(* CODESYS project plc_chalet_base.library
   Title: CHALET_BaseComponents
   Version: 3.6.9
   Placeholder: CHALET_BaseComponents
   Company: Beckhoff CH

Project tree, tasks and I/O mapping:
  libraries: Tc2_EtherCAT, * (Beckhoff Automation GmbH); Tc2_Standard, * (Beckhoff Automation GmbH); Tc2_System, * (Beckhoff Automation GmbH); Tc2_Utilities, * (Beckhoff Automation GmbH); Tc3_EventLogger, * (Beckhoff Automation GmbH); Tc3_Module, * (Beckhoff Automation GmbH)
  COMPONENTs/
    CoE-Access/
      internal/
        function block FB_CoE_Base [ST]: cbBufLen, Index, pSrcBuf, SubIndex, Error, FB_init, ReadDone, Update, WriteDone
        interface I_AdsAddr: NetId, Port
      function block FB_CoE_BOOL [ST]: cbBufLen, pSrcBuf, Value
      function block FB_CoE_BYTE [ST]: cbBufLen, pSrcBuf, Value
      function block FB_CoE_Connection [ST]: Mapped, NetId, Port
      function block FB_CoE_UDINT [ST]: cbBufLen, pSrcBuf, Value
      function block FB_CoE_UINT [ST]: cbBufLen, pSrcBuf, Value
    EtherCatDiag/
      Subobject/
        data type E_EtherCatState
        function block FB_EtherCatSlaveDiag [ST]: AlarmHandling, DeviceAmsAddr, DeviceType, Name, SetConfig, State, StateBits, Update
        interface I_EtherCatSlaveDiag: DeviceAmsAddr, DeviceType, Name, State, StateBits
      function block FB_EtherCatMasterDiag [ST]: Initialize, Initialized, ListOfDevices, Mapped, NumerOfDevice, Update
      data type ST_XtsMotorEtherCatDiag
    Feedback/
      function block FB_CH_Feedback [ST]: ActiveCommand, Busy, Done, Error, ErrorId, FB_init, HR, LastCommandAccepted, UpdateEventlogger
      interface I_CH_Feedback: ActiveCommand, Busy, Done, Error, ErrorId, HR, LastCommandAccepted
    HR/
      function CheckNotOk [ST]
      function CheckOk [ST]
      function GetMostSignificant [ST]
    List/
      CD_CH_List
      function block FB_CH_List [ST]: Content, FindLUID, FindOID, FindOIDString, LUIDInList, OIDInList, ResetIterator, RestoreIterator, AddList, Clear, Duplicate, Initialize, IsEmpty, IsFull, Size, Update, AddObject, GetNextObject, GetRandomObject, HasNextObject, ObjectInList, RemoveAllDuplicateObjects, RemoveObject, GetObjectWithHighestNumber, GetObjectWithLowestNumber, Sort
      interface I_CH_List: Content, FindLUID, FindOID, FindOIDString, LUIDInList, OIDInList, ResetIterator, RestoreIterator, IsEmpty, IsFull, Size, GetNextObject, GetRandomObject, HasNextObject, ObjectInList, RemoveAllDuplicateObjects, GetObjectWithHighestNumber, GetObjectWithLowestNumber
      interface I_CH_List_Dublicate: Content
    Object/
      CD_CH_Object
      function block FB_CH_Object [ST]: FB_init, Initialize, LUID, OID, SortOrderInList, TaskIndex, Update
      interface I_CH_Object: Initialize, LUID, OID, SortOrderInList, Update
    function F_Convert32InPastTo64Bit [ST]
  CONSTANTs/
    data type E_Colors_ARGB
    global variables GVL_Datatypes
  global variables BaseParameterlist
  00000000-0000-0000-0000-000000000000|LICENSE.md
  LICENSE.md
*)

// COMPONENTs/EtherCatDiag/Subobject/E_EtherCatState
{attribute 'qualified_only'}
{attribute 'strict'}
{attribute 'to_string'}
TYPE E_EtherCatState :
(
	Unknown,
	Init,
	PreOp,
	BootStrap,
	SafeOp,
	Op,
	Disabled,
	Error
) := Unknown ;
END_TYPE

// COMPONENTs/EtherCatDiag/ST_XtsMotorEtherCatDiag
TYPE ST_XtsMotorEtherCatDiag :
STRUCT
	fbSource : FB_TcSourceInfo;
	fbAlarmNotInOpMode : FB_TcAlarm;
	fbAlarmNoCommunication : FB_TcAlarm;
	
	fbGetSlaveState : FB_EcGetSlaveState;
	nLastState : BYTE;
END_STRUCT
END_TYPE

// CONSTANTs/E_Colors_ARGB
{attribute 'qualified_only'}
{attribute 'strict'}
{attribute 'to_string'}
TYPE E_Colors_ARGB : (
        Darkred              := 16#FF8B0000, // rgb(139,0,0)
        Brown                := 16#FFA52A2A, // rgb(165,42,42)
        Firebrick            := 16#FFB22222, // rgb(178,34,34)
        Crimson              := 16#FFDC143C, // rgb(220,20,60)
        Red                  := 16#FFFF0000, // rgb(255,0,0)
        Tomato               := 16#FFFF6347, // rgb(255,99,71)
        Coral                := 16#FFFF7F50, // rgb(255,127,80)
        Indianred            := 16#FFCD5C5C, // rgb(205,92,92)
        Lightcoral           := 16#FFF08080, // rgb(240,128,128)
        Darksalmon           := 16#FFE9967A, // rgb(233,150,122)
        Salmon               := 16#FFFA8072, // rgb(250,128,114)
        Lightsalmon          := 16#FFFFA07A, // rgb(255,160,122)
        Orangered            := 16#FFFF4500, // rgb(255,69,0)
        Darkorange           := 16#FFFF8C00, // rgb(255,140,0)
        Orange               := 16#FFFFA500, // rgb(255,165,0)
        Gold                 := 16#FFFFD700, // rgb(255,215,0)
        Darkgoldenrod        := 16#FFB8860B, // rgb(184,134,11)
        Goldenrod            := 16#FFDAA520, // rgb(218,165,32)
        Palegoldenrod        := 16#FFEEE8AA, // rgb(238,232,170)
        Darkkhaki            := 16#FFBDB76B, // rgb(189,183,107)
        Khaki                := 16#FFF0E68C, // rgb(240,230,140)
        Olive                := 16#FF808000, // rgb(128,128,0)
        Yellow               := 16#FFFFFF00, // rgb(255,255,0)
        Yellowgreen          := 16#FF9ACD32, // rgb(154,205,50)
        Darkolivegreen       := 16#FF556B2F, // rgb(85,107,47)
        Olivedrab            := 16#FF6B8E23, // rgb(107,142,35)
        Lawngreen            := 16#FF7CFC00, // rgb(124,252,0)
        Chartreuse           := 16#FF7FFF00, // rgb(127,255,0)
        Greenyellow          := 16#FFADFF2F, // rgb(173,255,47)
        Darkgreen            := 16#FF006400, // rgb(0,100,0)
        Green                := 16#FF008000, // rgb(0,128,0)
        Forestgreen          := 16#FF228B22, // rgb(34,139,34)
        Lime                 := 16#FF00FF00, // rgb(0,255,0)
        Limegreen            := 16#FF32CD32, // rgb(50,205,50)
        Lightgreen           := 16#FF90EE90, // rgb(144,238,144)
        Palegreen            := 16#FF98FB98, // rgb(152,251,152)
        Darkseagreen         := 16#FF8FBC8F, // rgb(143,188,143)
        Mediumspringgreen    := 16#FF00FA9A, // rgb(0,250,154)
        Springgreen          := 16#FF00FF7F, // rgb(0,255,127)
        Seagreen             := 16#FF2E8B57, // rgb(46,139,87)
        Mediumaquamarine     := 16#FF66CDAA, // rgb(102,205,170)
        Mediumseagreen       := 16#FF3CB371, // rgb(60,179,113)
        Lightseagreen        := 16#FF20B2AA, // rgb(32,178,170)
        Darkslategray        := 16#FF2F4F4F, // rgb(47,79,79)
        Teal                 := 16#FF008080, // rgb(0,128,128)
        Darkcyan             := 16#FF008B8B, // rgb(0,139,139)
        Aqua                 := 16#FF00FFFF, // rgb(0,255,255)
        Lightcyan            := 16#FFE0FFFF, // rgb(224,255,255)
        Darkturquoise        := 16#FF00CED1, // rgb(0,206,209)
        Turquoise            := 16#FF40E0D0, // rgb(64,224,208)
        Mediumturquoise      := 16#FF48D1CC, // rgb(72,209,204)
        Paleturquoise        := 16#FFAFEEEE, // rgb(175,238,238)
        Aquamarine           := 16#FF7FFFD4, // rgb(127,255,212)
        Powderblue           := 16#FFB0E0E6, // rgb(176,224,230)
        Cadetblue            := 16#FF5F9EA0, // rgb(95,158,160)
        Steelblue            := 16#FF4682B4, // rgb(70,130,180)
        Cornflowerblue       := 16#FF6495ED, // rgb(100,149,237)
        Deepskyblue          := 16#FF00BFFF, // rgb(0,191,255)
        Dodgerblue           := 16#FF1E90FF, // rgb(30,144,255)
        Lightblue            := 16#FFADD8E6, // rgb(173,216,230)
        Skyblue              := 16#FF87CEEB, // rgb(135,206,235)
        Lightskyblue         := 16#FF87CEFA, // rgb(135,206,250)
        Midnightblue         := 16#FF191970, // rgb(25,25,112)
        Navy                 := 16#FF000080, // rgb(0,0,128)
        Darkblue             := 16#FF00008B, // rgb(0,0,139)
        Mediumblue           := 16#FF0000CD, // rgb(0,0,205)
        Blue                 := 16#FF0000FF, // rgb(0,0,255)
        Royalblue            := 16#FF4169E1, // rgb(65,105,225)
        Blueviolet           := 16#FF8A2BE2, // rgb(138,43,226)
        Indigo               := 16#FF4B0082, // rgb(75,0,130)
        Darkslateblue        := 16#FF483D8B, // rgb(72,61,139)
        Slateblue            := 16#FF6A5ACD, // rgb(106,90,205)
        Mediumslateblue      := 16#FF7B68EE, // rgb(123,104,238)
        Mediumpurple         := 16#FF9370DB, // rgb(147,112,219)
        Darkmagenta          := 16#FF8B008B, // rgb(139,0,139)
        Darkviolet           := 16#FF9400D3, // rgb(148,0,211)
        Darkorchid           := 16#FF9932CC, // rgb(153,50,204)
        Mediumorchid         := 16#FFBA55D3, // rgb(186,85,211)
        Purple               := 16#FF800080, // rgb(128,0,128)
        Thistle              := 16#FFD8BFD8, // rgb(216,191,216)
        Plum                 := 16#FFDDA0DD, // rgb(221,160,221)
        Violet               := 16#FFEE82EE, // rgb(238,130,238)
        Magenta              := 16#FFFF00FF, // rgb(255,0,255)
        Orchid               := 16#FFDA70D6, // rgb(218,112,214)
        Mediumvioletred      := 16#FFC71585, // rgb(199,21,133)
        Palevioletred        := 16#FFDB7093, // rgb(219,112,147)
        Deeppink             := 16#FFFF1493, // rgb(255,20,147)
        Hotpink              := 16#FFFF69B4, // rgb(255,105,180)
        Lightpink            := 16#FFFFB6C1, // rgb(255,182,193)
        Pink                 := 16#FFFFC0CB, // rgb(255,192,203)
        Antiquewhite         := 16#FFFAEBD7, // rgb(250,235,215)
        Beige                := 16#FFF5F5DC, // rgb(245,245,220)
        Bisque               := 16#FFFFE4C4, // rgb(255,228,196)
        Blanchedalmond       := 16#FFFFEBCD, // rgb(255,235,205)
        Wheat                := 16#FFF5DEB3, // rgb(245,222,179)
        Cornsilk             := 16#FFFFF8DC, // rgb(255,248,220)
        Lemonchiffon         := 16#FFFFFACD, // rgb(255,250,205)
        LightGoldenRodYellow := 16#FFFAFAD2, // rgb(250,250,210)
        LightYellow          := 16#FFFFFFE0, // rgb(255,255,224)
        SaddleBrown          := 16#FF8B4513, // rgb(139,69,19)
        Sienna               := 16#FFA0522D, // rgb(160,82,45)
        Chocolate            := 16#FFD2691E, // rgb(210,105,30)
        Peru                 := 16#FFCD853F, // rgb(205,133,63)
        SandyBrown           := 16#FFF4A460, // rgb(244,164,96)
        BurlyWood            := 16#FFDEB887, // rgb(222,184,135)
        RosyBrown            := 16#FFBC8F8F, // rgb(188,143,143)
        Moccasin             := 16#FFFFE4B5, // rgb(255,228,181)
        NavajoWhite          := 16#FFFFDEAD, // rgb(255,222,173)
        PeachPuff            := 16#FFFFDAB9, // rgb(255,218,185)
        MistyRose            := 16#FFFFE4E1, // rgb(255,228,225)
        LavenderBlush        := 16#FFFFF0F5, // rgb(255,240,245)
        Linen                := 16#FFFAF0E6, // rgb(250,240,230)
        OldLace              := 16#FFFDF5E6, // rgb(253,245,230)
        PapayaWhip           := 16#FFFFEFD5, // rgb(255,239,213)
        Seashell             := 16#FFFFF5EE, // rgb(255,245,238)
        MintCream            := 16#FFF5FFFA, // rgb(245,255,250)
        SlateGray            := 16#FF708090, // rgb(112,128,144)
        LightSlateGray       := 16#FF778899, // rgb(119,136,153)
        LightSteelBlue       := 16#FFB0C4DE, // rgb(176,196,222)
        Lavender             := 16#FFE6E6FA, // rgb(230,230,250)
        FloralWhite          := 16#FFFFFAF0, // rgb(255,250,240)
        AliceBlue            := 16#FFF0F8FF, // rgb(240,248,255)
        GhostWhite           := 16#FFF8F8FF, // rgb(248,248,255)
        HoneyDew             := 16#FFF0FFF0, // rgb(240,255,240)
        Ivory                := 16#FFFFFFF0, // rgb(255,255,240)
        Azure                := 16#FFF0FFFF, // rgb(240,255,255)
        Snow                 := 16#FFFFFAFA, // rgb(255,250,250)
        Black                := 16#FF000000, // rgb(0,0,0)
        DimGray              := 16#FF696969, // rgb(105,105,105)
        Gray                 := 16#FF808080, // rgb(128,128,128)
        DarkGray             := 16#FFA9A9A9, // rgb(169,169,169)
        Silver               := 16#FFC0C0C0, // rgb(192,192,192)
        LightGray            := 16#FFD3D3D3, // rgb(211,211,211)
        Gainsboro            := 16#FFDCDCDC, // rgb(220,220,220)
        WhiteSmoke           := 16#FFF5F5F5, // rgb(245,245,245)
        White                := 16#FFFFFFFF  // rgb(255,255,255)
    ) UDINT;
END_TYPE

// CONSTANTs/GVL_Datatypes
{attribute 'qualified_only'}
VAR_GLOBAL CONSTANT
	// SINT
	cMaxSint	: SINT 		:= 127; // Largest SINT number
    cMinSint	: SINT 		:= -128; // Smallest SINT number

	// USINT
	cMaxUsint	: USINT 	:= 255; // Largest USINT number
    cMinUSint	: USINT 	:= 0; // Smallest USINT number

	// INT
	cMaxInt		: INT 		:= 32_767; // Largest INT number
    cMinInt		: INT 		:= -32_768; // Smallest INT number

	// UINT
	cMaxUint	: UINT 		:= 65_535; // Largest UINT number
    cMinUnit	: UINT 		:= 0; // Smallest UINT number

	// DINT
	cMaxDint	: DINT 		:= 2_147_483_647; // Largest DINT number
    cMinDint	: DINT 		:= -2_147_483_648; // Smallest DINT number

	// UDINT
	cMaxUdint	: UDINT 	:= 4_294_967_295; // Largest UDINT number
    cMinUdint	: UDINT		:= 0; // Smallest UDINT number

	// LINT
	cMaxLint	: LINT 		:= 9_223_372_036_854_775_807; // Largest LINT number
    cMinBLint	: LINT 		:= -9_223_372_036_854_775_808; // Smallest LINT number

	// ULINT
	cMaxUlint	: ULINT 	:= 18_446_744_073_709_551_615; // Largest ULINT number
    cMinUlint	: ULINT 	:= 0; // Smallest ULINT number

	// BYTE
	cMaxByte	: BYTE 		:= 255; // Largest BYTE number
    cMinByte	: BYTE 		:= 0; // Smallest BYTE number

	// WORD
	cMaxWord	: WORD 		:= 65_535; // Largest WORD number
    cMinWord	: WORD 		:= 0; // Smallest WORD number

	// DWORD
	cMaxDword	: DWORD 	:= 4_294_967_295; // Largest DWORD number
    cMinDword	: DWORD 	:= 0; // Smallest DWORD number

	// LWORD
	cMaxLword	: LWORD 	:= 18_446_744_073_709_551_615; // Largest LWORD number
    cMinLword	: LWORD 	:= 0; // Smallest LWORD number
	
	// REAL
	cMaxReal	: REAL 		:= 3.402823E+38; // Largest REAL number
    cMinReal	: REAL 		:= -3.402823E+38; // Smallest REAL number
	
	// LREAL
    cMaxLreal	: LREAL 	:= 1.7976931348623157E+308; // Largest LREAL number
    cMinLreal	: LREAL 	:= -1.7976931348623157E+308; // Smallest LREAL number
	
    // DATE
    cMaxDate   	: DATE    	:= DATE#2106-2-7; // Maximum DATA
    cMinDate   	: DATE     	:= DATE#1970-1-1; // Minimum DATE
	
	// TIME
	cMaxTime	: TIME  	:= T#49D17H2M47S295MS; // Longest TIME duration
	cMinTime 	: TIME  	:= TO_TIME(0);	// Shortest TIME duration
	
	// LTIME
	cMaxLtime	: LTIME 	:= LTIME#213503D23H34M33S709MS551US615NS; // Longest LTIME duration
	cMinLtime 	: LTIME  	:= TO_LTIME(0); // Shortest LTIME duration
	
    // Date and time
    cMaxDataAndTime  : DATE_AND_TIME  := DATE_AND_TIME#2106-02-07-06:28:15; // Maximum DATA_AND_DATE
    cMinDataAndTime  : DATE_AND_TIME  := DATE_AND_TIME#1970-1-1-0:0:0; // Minimum DATA_AND_DATE

    // Time of day
    cMaxTimeOfDay 	: TIME_OF_DAY    := TIME_OF_DAY#23:59:59.999; // Largest TIME_OF_DAY
    cMinTimeOfDay 	: TIME_OF_DAY    := TIME_OF_DAY#0:0:0; // Smallest TIME_OF_DAY
END_VAR

// BaseParameterlist
{attribute 'qualified_only'}
VAR_GLOBAL CONSTANT
	(*Maximum length of FB_CH_Object*)
	MAX_OBJECTS 			: UDINT := 150;
	
	(*Maximum CoE-Read at same time*)
	MAX_COE_READ 			: UDINT := 20;
	
	(*Maximum CoE-Write at same time*)
	MAX_COE_WRITE 			: UDINT := 20;
	
	(*Write an info to the event logger when FB_Feedback is busy*)
	B_WRITE_INFO_FEEDBACK_BUSY 	: BOOL := TRUE;
	
END_VAR

// COMPONENTs/CoE-Access/internal/FB_CoE_Base
(* This FB is abstract and is the base class  *)
FUNCTION_BLOCK ABSTRACT FB_CoE_Base EXTENDS FB_CH_Object
VAR
	//Coe Connector
	{attribute 'hide'}
	ipCoeConnection	: I_AdsAddr;
	{attribute 'hide'}
	bErrorInvalideInterface : BOOL;
	
	//Parameter index
	{attribute 'hide'}
    nIndex     : WORD; (* CoE Object Index *)
	{attribute 'hide'}
    nSubIndex  : BYTE; (* Subindex of CoE Object *)

	//Read/write 
	{attribute 'hide'}
	bReadDone : BOOL;
	{attribute 'hide'}
	fbCoeRead : FB_EcCoeSdoRead;
	{attribute 'hide'}
	nSeqRead : UINT;
	{attribute 'hide'}
	bReadError : BOOL;
	
	{attribute 'hide'}
	bWriteDone : BOOL := TRUE;
	{attribute 'hide'}
	fbCoeWrite : FB_EcCoeSdoWrite;
	{attribute 'hide'}
	nSeqWrite : UINT;
	{attribute 'hide'}
	bWriteError : BOOL;
	
	{attribute 'hide'}
	fbDelayOnError : TON := ( PT:= T#10S);
END_VAR
VAR_STAT
	nCtsCoeObject : UDINT;
	nCtsReadActive : UDINT;
	nCtsWriteActive : UDINT;
END_VAR

PROPERTY PROTECTED ABSTRACT cbBufLen : UDINT
GET
END_GET
END_PROPERTY

PROPERTY PRIVATE Index : WORD
GET
END_GET
END_PROPERTY

PROPERTY PROTECTED ABSTRACT pSrcBuf : PVOID
GET
END_GET
END_PROPERTY

PROPERTY PRIVATE SubIndex : BYTE
GET
END_GET
END_PROPERTY

{attribute 'monitoring':='call'}
PROPERTY Error : BOOL
GET
Error := THIS^.bReadError OR THIS^.bWriteError OR THIS^.bErrorInvalideInterface;
END_GET
END_PROPERTY

METHOD FB_init : BOOL
VAR_INPUT
	bInitRetains : BOOL; // if TRUE, the retain variables are initialized (warm start / cold start)
	bInCopyCode : BOOL;  // if TRUE, the instance afterwards gets moved into the copy code (online change)
	
	ipCoeConnection	: I_AdsAddr;
    nIndex     : WORD; 	(* CoE Object Index *)
    nSubIndex  : BYTE; 		(* Subindex of CoE Object *)
END_VAR

VAR_INST
	{attribute 'hide'}
	bFBInitCalledOnce : BOOL; //Do the following code once during start up and not during onlinechange
END_VAR
//Do the following code once during start up and not during onlinechange
IF NOT bFBInitCalledOnce THEN 
	nCtsCoeObject := nCtsCoeObject +1;
	
	THIS^.ipCoeConnection := ipCoeConnection;
	THIS^.nIndex 		:= nIndex;
	THIS^.nSubIndex 	:= nSubIndex;
END_IF

bFBInitCalledOnce := TRUE;
END_METHOD

{attribute 'monitoring':='call'}
PROPERTY ReadDone : BOOL
GET
ReadDone := bReadDone;
END_GET
SET
//Only allow set to FALSE
IF NOT ReadDone THEN
	bReadDone := FALSE;
END_IF
END_SET
END_PROPERTY

METHOD Update : HRESULT
IF ipCoeConnection = 0 THEN
	bErrorInvalideInterface := TRUE;
	RETURN;
END_IF


(*--- Read ---*)
CASE nSeqRead OF
	0: //Start/Restart if required
		IF NOT bReadDone  AND bWriteDone(* Write has higher priority*) AND (nCtsReadActive < BaseParameterlist.MAX_COE_READ) AND (nSeqWrite = 0) THEN
			fbCoeRead.bExecute := TRUE; // Rising edge	
			nCtsReadActive := nCtsReadActive +1;	
			nSeqRead := 1;
		END_IF
	
	1: //Check if done or error
		IF fbCoeRead.bError THEN
			//Error
			nSeqRead := 99;
			bReadError := TRUE;
			fbDelayOnError.IN := TRUE;
			nCtsReadActive := nCtsReadActive -1;	
			
		ELSIF NOT fbCoeRead.bBusy AND NOT fbCoeRead.bError THEN
			//Done
			THIS^.bReadDone := TRUE;
			nSeqRead := 0;
			bReadError := FALSE;
			nCtsReadActive := nCtsReadActive -1;	
		END_IF	
		
	99: // Delay on error to reduce amount of errors
		IF fbDelayOnError.Q THEN
			fbDelayOnError.IN := FALSE;
			nSeqRead := 0;
		END_IF
END_CASE

IF NOT THIS^.bReadDone THEN
	fbCoeRead(
		sNetId		:= ipCoeConnection.NetId,
		nSlaveAddr	:= ipCoeConnection.port,
		nSubIndex	:= THIS^.nSubIndex, 
		nIndex		:= THIS^.nIndex, 
		pDstBuf		:= THIS^.pSrcBuf, 
		cbBufLen	:= THIS^.cbBufLen);
		
	//Prepare for next rising edge
	fbCoeRead.bExecute := FALSE;
END_IF



(*--- Write ---*)
CASE nSeqWrite OF
	0: //Start/Restart if required
		IF NOT bWriteDone AND (nCtsWriteActive < BaseParameterlist.MAX_COE_WRITE) AND (nSeqRead = 0) THEN
			fbCoeWrite.bExecute := TRUE; // Rising edge	
			nCtsWriteActive := nCtsWriteActive +1;	
			nSeqWrite := 1;
		END_IF
	
	1: //Check if done or error
		IF fbCoeWrite.bError THEN
			//Error
			nSeqWrite := 99;
			bWriteError := TRUE;
			fbDelayOnError.IN := TRUE;
			nCtsWriteActive := nCtsWriteActive -1;	
			
		ELSIF NOT fbCoeWrite.bBusy AND NOT fbCoeWrite.bError THEN
			//Done
			THIS^.bWriteDone := TRUE;
			nSeqWrite := 0;
			bWriteError := FALSE;
			nCtsWriteActive := nCtsWriteActive -1;	
		END_IF	
		
	99: // Delay on error to reduce amount of errors
		IF fbDelayOnError.Q THEN
			fbDelayOnError.IN := FALSE;
			nSeqWrite := 0;
		END_IF		

END_CASE

IF NOT bWriteDone THEN
	fbCoeWrite(
		sNetId		:= ipCoeConnection.netId, 
		nSlaveAddr	:= ipCoeConnection.port,
		nSubIndex	:= THIS^.nSubIndex, 
		nIndex		:= THIS^.nIndex, 
		pSrcBuf		:= THIS^.pSrcBuf, 
		cbBufLen	:= THIS^.cbBufLen);		
		
	//Prepare for next rising edge
	fbCoeWrite.bExecute := FALSE;
END_IF

//Update
fbDelayOnError();
END_METHOD

{attribute 'monitoring':='call'}
PROPERTY WriteDone : BOOL
GET
WriteDone := bWriteDone;
END_GET
SET
//Only allow set to FALSE
IF NOT WriteDone THEN
	bWriteDone := FALSE;
END_IF
END_SET
END_PROPERTY

END_FUNCTION_BLOCK

// COMPONENTs/Object/FB_CH_Object
FUNCTION_BLOCK FB_CH_Object IMPLEMENTS I_CH_Object
VAR
	(* The SourceInfo is created internally as the default behavior. 
	It then contains the symbol name of the function block that instances FB_TcMessage as SourceName and the object ID of the PLC instance as SourceID.
	If the instance of FB_TcMessage is hidden with the attribute "hide", no symbol name can be created internally for the default behavior. *)
	fbSourceInfo : FB_TcSourceInfo;
	
	{attribute 'hide'}
	nTaskIndex : BYTE; //Used in TwinCAT_SystemInfoVarList._TaskInfo	
	{attribute 'hide'}
	nSortOrderInList : UDINT; //Used in List in methode Sort()
END_VAR

METHOD FB_init : BOOL
VAR_INPUT
	bInitRetains : BOOL; // if TRUE, the retain variables are initialized (warm start / cold start)
	bInCopyCode : BOOL;  // if TRUE, the instance afterwards gets moved into the copy code (online change)
END_VAR
VAR
	fbGetCurTaskIdx  : GETCURTASKINDEX;
END_VAR
fbGetCurTaskIdx();
THIS^.nTaskIndex := fbGetCurTaskIdx.Index;
END_METHOD

METHOD Initialize : HRESULT
Initialize := S_OK;
END_METHOD

{attribute 'monitoring':='call'}
//Locally unique identifier
PROPERTY LUID : STRING
GET
LUID := THIS^.fbSourceInfo.sName;
END_GET
END_PROPERTY

{attribute 'monitoring':='call'}
//Unique object ID
PROPERTY OID : OTCID
GET
OID := 0;
END_GET
END_PROPERTY

//Optional. Is used in FB_CH_List in the “Sort()” method. The entire list is sorted by ascending number. (small numbers at the beginning)
PROPERTY SortOrderInList : UDINT
GET
SortOrderInList := nSortOrderInList;
END_GET
SET
nSortOrderInList := SortOrderInList;
END_SET
END_PROPERTY

//Used in TwinCAT_SystemInfoVarList._TaskInfo
PROPERTY PROTECTED TaskIndex : BYTE
GET
TaskIndex := THIS^.nTaskIndex;
END_GET
END_PROPERTY

METHOD Update : HRESULT
VAR_INPUT
END_VAR
Update := S_OK;
END_METHOD

END_FUNCTION_BLOCK

// COMPONENTs/Object/I_CH_Object
INTERFACE I_CH_Object EXTENDS __SYSTEM.IQueryInterface

METHOD Initialize : HRESULT
END_METHOD

{attribute 'monitoring':='call'}
//Locally unique identifier
PROPERTY LUID : STRING
GET
END_GET
END_PROPERTY

{attribute 'monitoring':='call'}
//Object ID
PROPERTY OID : OTCID
GET
END_GET
END_PROPERTY

//Optional. Is used in FB_CH_List in the “Sort()” method. The entire list is sorted by ascending number. (small numbers at the beginning)
PROPERTY SortOrderInList : UDINT
GET
END_GET
SET
END_SET
END_PROPERTY

METHOD Update : HRESULT
VAR_INPUT
END_VAR
END_METHOD

END_INTERFACE

// COMPONENTs/List/FB_CH_List
FUNCTION_BLOCK FB_CH_List EXTENDS FB_CH_Object IMPLEMENTS I_CH_LIST, I_CH_List_Dublicate
VAR
	{attribute 'hide'}
	nObjectCount			: UDINT;
	{attribute 'hide'}
	nIdxNextObject			: UDINT;
	{attribute 'hide'}
	nIdxLastRestoreValues : ARRAY [0..(MAX_CTS_RESTORE_VALUES+1)] OF UDINT;
	{attribute 'hide'}
	nIdxRestore				: UDINT;
	{attribute 'hide'}
	aObjects				: ARRAY [1..BaseParameterlist.MAX_OBJECTS] OF I_CH_Object;
END_VAR
VAR CONSTANT
	{attribute 'hide'}
	MAX_CTS_RESTORE_VALUES : UINT := 20;
END_VAR

//DEBUG only. View content for easy debug. Do not use this property
{attribute 'monitoring':='call'}
PROPERTY Content : REFERENCE TO ARRAY [1..BaseParameterlist.MAX_OBJECTS] OF I_CH_Object
GET
Content REF= THIS^.aObjects;
END_GET
END_PROPERTY

METHOD PUBLIC FindLUID : I_CH_OBJECT
VAR_INPUT
	sLUID	: STRING;
END_VAR
VAR
	nIdx : UDINT;
END_VAR
FOR nIdx := 1 TO nObjectCount DO
	IF aObjects[nIdx] <> 0 AND_THEN aObjects[nIdx].LUID = sLUID THEN
		FindLUID := aObjects[nIdx];
		EXIT;
	END_IF
END_FOR
END_METHOD

METHOD FindOID : I_CH_OBJECT
VAR_INPUT
	nOID	: OTCID;
END_VAR
VAR
	nIdx : UDINT;
END_VAR
FOR nIdx := 1 TO nObjectCount DO
	IF aObjects[nIdx] <> 0 AND_THEN aObjects[nIdx].OID = nOID THEN
		FindOID := aObjects[nIdx];
		EXIT;
	END_IF
END_FOR
END_METHOD

METHOD FindOIDString : I_CH_OBJECT
VAR_INPUT
	sOID	: STRING;
END_VAR
VAR
	nIdx : UDINT;
END_VAR
FOR nIdx := 1 TO nObjectCount DO
	IF aObjects[nIdx] <> 0 AND_THEN DWORD_TO_HEXSTR(TO_DWORD(aObjects[nIdx].OID),0,FALSE) = sOID THEN
		FindOIDString := aObjects[nIdx];
		EXIT;
	END_IF
END_FOR
END_METHOD

METHOD PUBLIC LUIDInList : BOOL
VAR_INPUT
	sLUID	: STRING;
END_VAR
VAR
	nIdx : UDINT;
END_VAR
//Check array until a match
FOR nIdx := 1 TO THIS^.nObjectCount DO
	IF THIS^.aObjects[nIdx].LUID = sLUID THEN
		LUIDInList := TRUE;
		EXIT;
	END_IF
END_FOR
END_METHOD

METHOD PUBLIC OIDInList : BOOL
VAR_INPUT
	nOID	: OTCID;
END_VAR
VAR
	nIdx : UDINT;
END_VAR
//Check array until a match
FOR nIdx := 1 TO THIS^.nObjectCount DO
	IF THIS^.aObjects[nIdx].OID = nOID THEN
		OIDInList := TRUE;
		EXIT;
	END_IF
END_FOR
END_METHOD

METHOD PUBLIC ResetIterator : BOOL
VAR_INPUT
END_VAR
//Store the last few index for later restore if required - Shift array +1 step
MEMMOVE(srcAddr 	:= ADR(nIdxLastRestoreValues[0]), 
		destAddr 	:= ADR(nIdxLastRestoreValues[1]), 
		n 			:= (SIZEOF(nIdxNextObject)*MAX_CTS_RESTORE_VALUES));

//Store the last few index for later restore if required - Store last value
nIdxLastRestoreValues[0] := nIdxNextObject;


nIdxNextObject := 0;
END_METHOD

//Restore the iterator to the value before the last reset. This is necessary if several while loops are placed inside each other
METHOD PUBLIC RestoreIterator : BOOL
VAR_INPUT
END_VAR
//Store the last few index for later restore if required - Restore
nIdxNextObject := nIdxLastRestoreValues[0];

//Store the last few index for later restore if required - Shift array -1 step
MEMMOVE(srcAddr 	:= ADR(nIdxLastRestoreValues[1]), 
		destAddr 	:= ADR(nIdxLastRestoreValues[0]), 
		n 			:= (SIZEOF(nIdxNextObject)*MAX_CTS_RESTORE_VALUES));
END_METHOD

//Add all objects from the list in to this list
METHOD PUBLIC AddList : HRESULT
VAR_INPUT
	ipList	: I_CH_List;
END_VAR
VAR
	hr : HRESULT;
	ipListDublicate : I_CH_List_Dublicate;
	refRemoteList : REFERENCE TO ARRAY [1..BaseParameterlist.MAX_OBJECTS] OF I_CH_Object;
	pRemoteList : PVOID;
END_VAR
VAR_INST
	{attribute 'hide'}
	fbAlarmInvalideInputparm : FB_TcAlarm;
	{attribute 'hide'}
	fbAlarmListToSmall : FB_TcAlarm;
END_VAR
// Invalide input
IF ipList = 0 THEN
	fbAlarmInvalideInputparm.CreateEx(stEventEntry:= TC_EVENTS.CHALET_Base_Events.Invalide_Inputparameter, 
							ipSourceInfo := THIS^.fbSourceInfo, 
							bWithConfirmation := FALSE);
	fbAlarmInvalideInputparm.ipArguments.Clear().AddStringByValue('ipList');
	fbAlarmInvalideInputparm.Raise(0);	

	AddList := S_FALSE;
	RETURN;
END_IF


// This list is to small
IF (ipList.Size + THIS^.Size) > BaseParameterlist.MAX_OBJECTS THEN
	fbAlarmListToSmall.CreateEx(stEventEntry:= TC_EVENTS.CHALET_Base_Events.ListIsToSmall, 
							ipSourceInfo := THIS^.fbSourceInfo, 
							bWithConfirmation := FALSE);
	fbAlarmListToSmall.Raise(0);	

	AddList := S_FALSE;
	RETURN;
END_IF


//Done nothing to add
IF ipList.Size = 0 THEN
	AddList := S_OK;
	RETURN;
END_IF


//Check if the list has an optional I_CH_List_Dublicate interface. If so use the faste memcpy, else use default list commands
IF __QUERYINTERFACE(ipList, ipListDublicate) AND_THEN __ISVALIDREF(ipListDublicate.Content) THEN
	refRemoteList REF= ipListDublicate.Content;
	pRemoteList := ADR(refRemoteList);
	Tc2_System.MEMCPY(destAddr:= ADR(THIS^.aObjects[(THIS^.nObjectCount+1)]), srcAddr:= pRemoteList, n:= (SIZEOF(THIS^.aObjects[1])*ipList.Size) );
	THIS^.nObjectCount := ipList.Size + THIS^.nObjectCount; //Set size of List
ELSE
	ipList.ResetIterator();
	WHILE ipList.HasNextObject() DO
		hr := THIS^.AddObject(ipList.GetNextObject());
		IF hr <> S_OK THEN
			//Error
			AddList := hr;
			RETURN;
		END_IF
	END_WHILE
	ipList.RestoreIterator();
END_IF
END_METHOD

METHOD PUBLIC Clear : BOOL
VAR
	nIdx : UDINT;
END_VAR
Tc2_System.MEMSET(	destAddr	:= ADR(aObjects[1]), 
					fillByte	:= 0, 
					n			:= SIZEOF(aObjects[1])*BaseParameterlist.MAX_OBJECTS);


nObjectCount	:= 0;
nIdxNextObject	:= 0;
END_METHOD

METHOD Duplicate : BOOL
VAR_INPUT
	ipListCopyFrom : I_CH_LIST;
END_VAR
VAR
	ipThisList : I_CH_LIST := THIS^;
	hr : HRESULT;
	ipListDublicate : I_CH_List_Dublicate;
	refRemoteList : REFERENCE TO ARRAY [1..BaseParameterlist.MAX_OBJECTS] OF I_CH_Object;
	pRemoteList : PVOID;
END_VAR
VAR_INST
	{attribute 'hide'}
	fbAlarmInvalideInputparm : FB_TcAlarm;
	{attribute 'hide'}
	fbAlarmListToSmall : FB_TcAlarm;
END_VAR
//New list equals this list
IF ipListCopyFrom = ipThisList THEN
	//Do Nothing - Successfull
	Duplicate := TRUE;
	RETURN;
END_IF

THIS^.Clear();

// Invalide input
IF ipListCopyFrom = 0 THEN
	fbAlarmInvalideInputparm.CreateEx(stEventEntry:= TC_EVENTS.CHALET_Base_Events.Invalide_Inputparameter, 
							ipSourceInfo := THIS^.fbSourceInfo, 
							bWithConfirmation := FALSE);
	fbAlarmInvalideInputparm.ipArguments.Clear().AddStringByValue('ipListCopyFrom');
	fbAlarmInvalideInputparm.Raise(0);	

	Duplicate := FALSE;
	RETURN;
END_IF


// This list is to small
IF ipListCopyFrom.Size > BaseParameterlist.MAX_OBJECTS THEN
	fbAlarmListToSmall.CreateEx(stEventEntry:= TC_EVENTS.CHALET_Base_Events.ListIsToSmall, 
							ipSourceInfo := THIS^.fbSourceInfo, 
							bWithConfirmation := FALSE);
	fbAlarmListToSmall.Raise(0);	
	Duplicate := FALSE;
	RETURN;
END_IF


//Done nothing to add
IF ipListCopyFrom.Size = 0 THEN
	Duplicate := TRUE;
	RETURN;
END_IF


//Check if the list has an optional I_CH_List_Dublicate interface. If so use the faste memcpy, else use list commands
IF __QUERYINTERFACE(ipListCopyFrom, ipListDublicate) AND_THEN __ISVALIDREF(ipListDublicate.Content) THEN
	refRemoteList REF= ipListDublicate.Content;
	pRemoteList := ADR(refRemoteList);
	Tc2_System.MEMCPY(destAddr:= ADR(THIS^.aObjects), srcAddr:= pRemoteList, n:= (SIZEOF(THIS^.aObjects[1])*ipListCopyFrom.Size) );
	THIS^.nObjectCount := ipListCopyFrom.Size; //Set size of List
ELSE
	ipListCopyFrom.ResetIterator();
	WHILE ipListCopyFrom.HasNextObject() DO
		hr := THIS^.AddObject(ipListCopyFrom.GetNextObject());
		IF hr <> S_OK THEN
			//Error
			Duplicate := FALSE;
			RETURN;
		END_IF
	END_WHILE
	ipListCopyFrom.RestoreIterator();	
END_IF


Duplicate := TRUE;
END_METHOD

METHOD Initialize : HRESULT //This method calls the respective Initialize method of all contained objects
VAR_INPUT
END_VAR
VAR
	hr : HRESULT;
	nIdx : UDINT;
END_VAR
//FOR each element
FOR nIdx := 1 TO nObjectCount DO
	// DO Init
	hr := GetMostSignificant(hr, aObjects[nIdx].Initialize());
END_FOR


Initialize := hr;
END_METHOD

{attribute 'monitoring':='call'}
PROPERTY PUBLIC IsEmpty : BOOL
GET
IsEmpty := (nObjectCount = 0);
END_GET
END_PROPERTY

{attribute 'monitoring':='call'}
PROPERTY PUBLIC IsFull : BOOL
GET
IsFull := (nObjectCount = BaseParameterlist.MAX_OBJECTS);
END_GET
END_PROPERTY

{attribute 'monitoring':='call'}
PROPERTY PUBLIC Size : UDINT
GET
Size := nObjectCount;
END_GET
END_PROPERTY

METHOD Update : HRESULT //This method calls the respective update method of all contained objects
VAR
	hr : HRESULT;
	nIdx : UDINT;
END_VAR
//FOR each element
FOR nIdx := 1 TO nObjectCount DO
	// DO Update
	hr := GetMostSignificant(hr, aObjects[nIdx].Update());
END_FOR

Update := hr;
END_METHOD

METHOD PUBLIC AddObject : HRESULT
VAR_INPUT
	iChObject	: I_CH_Object;
END_VAR
VAR_INST
	{attribute 'hide'}
	fbAlarmListFull : FB_TcAlarm;
END_VAR
IF iChObject = 0 THEN
	AddObject := S_FALSE;
	RETURN;
END_IF


//Error if list is allready full
IF nObjectCount >= BaseParameterlist.MAX_OBJECTS THEN
	fbAlarmListFull.CreateEx(stEventEntry:= TC_EVENTS.CHALET_Base_Events.ListIsFull, 
							ipSourceInfo := THIS^.fbSourceInfo, 
							bWithConfirmation := FALSE);
	fbAlarmListFull.ipArguments.Clear().AddStringByValue(iChObject.LUID);
	fbAlarmListFull.Raise(0);
	AddObject := S_FALSE;
	RETURN;
END_IF


//Add to list
nObjectCount := nObjectCount + 1;
aObjects[nObjectCount] := iChObject;

AddObject := S_OK;
END_METHOD

METHOD PUBLIC GetNextObject : I_CH_Object
VAR_INPUT
END_VAR
VAR_INST
	{attribute 'hide'}
	fbAlarmInvalideEndOfList : FB_TcAlarm;
END_VAR
nIdxNextObject := nIdxNextObject + 1;


IF nIdxNextObject > nObjectCount THEN
	//Error!
	fbAlarmInvalideEndOfList.CreateEx(stEventEntry:= TC_EVENTS.CHALET_Base_Events.Invalive_EndOfList, 
							ipSourceInfo := THIS^.fbSourceInfo, 
							bWithConfirmation := FALSE);
	fbAlarmInvalideEndOfList.ipArguments.Clear().AddStringByValue('.GetNextObject()');
	fbAlarmInvalideEndOfList.Raise(0);
	RETURN;
END_IF




GetNextObject := aObjects[nIdxNextObject];
END_METHOD

METHOD GetRandomObject : I_CH_Object
VAR_INPUT
END_VAR

VAR_INST
	{attribute 'hide'}
	fbDRAN : DRAND;
END_VAR

VAR
	nRandomIdx : UDINT;
END_VAR
//Check if not Empty
IF UDINT_TO_BOOL(nObjectCount) THEN
	// Generate number 0..1
	fbDRAN(Seed:= 42);
	
	// 1..Size   = ((0..1)*(Size-1))+1
	nRandomIdx := LREAL_TO_UDINT(fbDRAN.Num * (nObjectCount-1))+1;
	
	GetRandomObject := aObjects[nRandomIdx];
	
END_IF
END_METHOD

METHOD PUBLIC HasNextObject : BOOL
VAR_INPUT
END_VAR
HasNextObject := (nIdxNextObject < nObjectCount) AND_THEN (aObjects[nIdxNextObject+1] <> 0);
END_METHOD

METHOD PUBLIC ObjectInList : BOOL
VAR_INPUT
	iChObject	: I_CH_Object;
END_VAR
VAR
	nIdx : UDINT;
END_VAR
//Check array until a match
FOR nIdx := 1 TO THIS^.nObjectCount DO
	IF THIS^.aObjects[nIdx] = iChObject THEN
		ObjectInList := TRUE;
		EXIT;
	END_IF
END_FOR
END_METHOD

METHOD RemoveAllDuplicateObjects : HRESULT
VAR_INPUT
END_VAR
VAR
	nIdx : UDINT;
	fbTempList : FB_CH_List;
	fbFoundDublicateObjects : FB_CH_List;
END_VAR
//Check eacht element in array, if allready was added in temp list. if found, delete
FOR nIdx := 1 TO THIS^.nObjectCount DO
	
	//check if allready was found
	IF fbTempList.ObjectInList(THIS^.aObjects[nIdx]) THEN
		//Found, add to an list to delete in next step
		fbFoundDublicateObjects.AddObject(THIS^.aObjects[nIdx]);	
	ELSE
		//Not found, add to list
		fbTempList.AddObject(THIS^.aObjects[nIdx]);	
	END_IF
END_FOR


//Delete in this list
fbFoundDublicateObjects.ResetIterator();
WHILE fbFoundDublicateObjects.HasNextObject() DO
	THIS^.RemoveObject(fbFoundDublicateObjects.GetNextObject());
END_WHILE
END_METHOD

METHOD PUBLIC RemoveObject : BOOL
VAR_INPUT
	iChObject	: I_CH_Object;
END_VAR

VAR
	nIdx			: UDINT;
END_VAR
RemoveObject := FALSE;

IF iChObject = 0 THEN
	RETURN;
END_IF

IF NOT THIS^.ObjectInList(iChObject) THEN
	RETURN;
END_IF

FOR nIdx := 1 TO nObjectCount DO
	IF aObjects[nIdx] = iChObject THEN
		aObjects[nIdx] := NULL;	
		
		nObjectCount := nObjectCount - 1;
		
		// Fill up the empty slot
		MEMMOVE(ADR(aObjects[nIdx]), ADR(aObjects[nIdx + 1]), SIZEOF(aObjects[nIdx]) * (BaseParameterlist.MAX_OBJECTS - nIdx));
	
		// If pos in list is less than ListIterator, then reduce Iterator
		IF nIdx <= nIdxNextObject THEN
			nIdxNextObject := nIdxNextObject -1;
		END_IF
		
		//Finish
		RemoveObject := TRUE;
		EXIT;
			
	END_IF
END_FOR
END_METHOD

METHOD GetObjectWithHighestNumber : I_CH_Object

VAR
	nIdx : UDINT;
	nMaxSortNbr : UDINT;
END_VAR




//Check array until a match
FOR nIdx := 1 TO THIS^.nObjectCount DO
	IF THIS^.aObjects[nIdx].SortOrderInList >= nMaxSortNbr THEN
		GetObjectWithHighestNumber := THIS^.aObjects[nIdx];
		nMaxSortNbr := THIS^.aObjects[nIdx].SortOrderInList;
	END_IF
END_FOR
END_METHOD

METHOD GetObjectWithLowestNumber : I_CH_Object
VAR
	nIdx : UDINT;
	nMinSortNbr : UDINT := GVL_Datatypes.cMaxUDint;
END_VAR
//Check array until a match
FOR nIdx := 1 TO THIS^.nObjectCount DO
	IF THIS^.aObjects[nIdx].SortOrderInList <= nMinSortNbr THEN
		GetObjectWithLowestNumber := THIS^.aObjects[nIdx];
		nMinSortNbr := THIS^.aObjects[nIdx].SortOrderInList;
	END_IF
END_FOR
END_METHOD

//Tthe entire list sorted BY ascending number. (small numbers AT the beginning).
//The FB_CH_Object.SortOrderInList is used
METHOD Sort : HRESULT
VAR
	fbCopyOfList : FB_CH_List;
	ipObjToAdd : I_CH_Object;
END_VAR
//TODO: use a smarter algorithm with less computational effort




//Create a copy of this list
fbCopyOfList.Duplicate(THIS^);

//Clear this List
THIS^.Clear();

//Add the smalest number to this list
WHILE NOT fbCopyOfList.IsEmpty DO
	ipObjToAdd := fbCopyOfList.GetObjectWithLowestNumber();
	fbCopyOfList.RemoveObject(ipObjToAdd);
	THIS^.AddObject(ipObjToAdd);
END_WHILE
END_METHOD

END_FUNCTION_BLOCK

// COMPONENTs/List/I_CH_List
INTERFACE I_CH_List EXTENDS __SYSTEM.IQueryInterface

//DEBUG only. View content for easy debug. Do not use this property
{attribute 'monitoring':='call'}
PROPERTY Content : REFERENCE TO ARRAY [1..BaseParameterlist.MAX_OBJECTS] OF I_CH_Object
GET
END_GET
END_PROPERTY

METHOD PUBLIC FindLUID : I_CH_OBJECT
VAR_INPUT
	sLUID	: STRING;
END_VAR
END_METHOD

METHOD FindOID : I_CH_OBJECT
VAR_INPUT
	nOID	: OTCID;
END_VAR
END_METHOD

METHOD FindOIDString : I_CH_OBJECT
VAR_INPUT
	sOID	: STRING;
END_VAR
END_METHOD

METHOD PUBLIC LUIDInList : BOOL
VAR_INPUT
	sLUID	: STRING;
END_VAR
END_METHOD

METHOD PUBLIC OIDInList : BOOL
VAR_INPUT
	nOID	: OTCID;
END_VAR
END_METHOD

METHOD PUBLIC ResetIterator : BOOL
VAR_INPUT
END_VAR
END_METHOD

//Restore the iterator to the value before the last reset. This is necessary if several while loops are placed inside each other
METHOD PUBLIC RestoreIterator : BOOL
VAR_INPUT
END_VAR
END_METHOD

{attribute 'monitoring':='call'}
PROPERTY PUBLIC IsEmpty : BOOL
GET
END_GET
END_PROPERTY

{attribute 'monitoring':='call'}
PROPERTY PUBLIC IsFull : BOOL
GET
END_GET
END_PROPERTY

{attribute 'monitoring':='call'}
PROPERTY PUBLIC Size : UDINT
GET
END_GET
END_PROPERTY

METHOD PUBLIC GetNextObject : I_CH_Object
VAR_INPUT
END_VAR
END_METHOD

METHOD GetRandomObject : I_CH_Object
VAR_INPUT
END_VAR
END_METHOD

METHOD PUBLIC HasNextObject : BOOL
VAR_INPUT
END_VAR
END_METHOD

METHOD PUBLIC ObjectInList : BOOL
VAR_INPUT
	iChObject	: I_CH_Object;
END_VAR
END_METHOD

METHOD RemoveAllDuplicateObjects : HRESULT
VAR_INPUT
END_VAR
END_METHOD

METHOD GetObjectWithHighestNumber : I_CH_Object
END_METHOD

METHOD GetObjectWithLowestNumber : I_CH_Object
END_METHOD

END_INTERFACE

// COMPONENTs/List/I_CH_List_Dublicate
INTERFACE I_CH_List_Dublicate EXTENDS __SYSTEM.IQueryInterface

{attribute 'monitoring':='call'}
PROPERTY Content : REFERENCE TO ARRAY [1..BaseParameterlist.MAX_OBJECTS] OF I_CH_Object
GET
END_GET
END_PROPERTY

END_INTERFACE

// COMPONENTs/HR/GetMostSignificant
(*
	Return the most significant HRESULT input (hr1 or hr2).
	Example: if hr1:= S_Pending and hr2 := S_OK, then return S_Pending 
	Priority:(Error(incl. code) > Error(empty code) > S_WATCHDOGTIMEOUT > S_PENDING > S_FALSE > S_OK)
*)
FUNCTION GetMostSignificant : HRESULT
VAR_INPUT
	hr1 : HRESULT; //top priority if both hr1 and hr2 have an error code return this
	hr2 : HRESULT; //second priority if both hr1 and hr2 have an error code return hr1
END_VAR

//hr1 has an Error(incl. errorcode) 
IF hr1.31 AND ((TO_DWORD(hr1) AND 16#FFF) > 0) THEN
	GetMostSignificant := hr1;

//hr2 has an Error(incl. errorcode) 
ELSIF hr2.31 AND ((TO_DWORD(hr2) AND 16#FFF) > 0) THEN
	GetMostSignificant := hr2;

//hr1 has an Error(empty errorcode)
ELSIF hr1.31 THEN
	GetMostSignificant := hr1;

//hr2 has an Error(empty errorcode)
ELSIF hr2.31 THEN
	GetMostSignificant := hr2;
	
//hr1 has a higher SUCCESS code than hr2. (S_WATCHDOGTIMEOUT > S_PENDING > S_FALSE > S_OK)
ELSIF hr1 >= hr2 THEN
	GetMostSignificant := hr1;

//hr2 has a higher SUCCESS code than hr1. (S_WATCHDOGTIMEOUT > S_PENDING > S_FALSE > S_OK)
ELSE 
	GetMostSignificant := hr2;	
	
END_IF

END_FUNCTION

// COMPONENTs/CoE-Access/internal/I_AdsAddr
INTERFACE I_AdsAddr

{attribute 'monitoring':='call'}
PROPERTY NetId : T_AmsNetID
GET
END_GET
END_PROPERTY

{attribute 'monitoring':='call'}
PROPERTY Port : WORD
GET
END_GET
END_PROPERTY

END_INTERFACE

// COMPONENTs/CoE-Access/FB_CoE_BOOL
{attribute 'no_explicit_call' := 'Do not call the body - Stick to OOP'}
FUNCTION_BLOCK FB_CoE_BOOL EXTENDS FB_CoE_Base
VAR
	{attribute 'hide'}
	nValue : BOOL;
END_VAR

PROPERTY PROTECTED cbBufLen : UDINT
GET
cbBufLen := SIZEOF(nValue);
END_GET
END_PROPERTY

PROPERTY PROTECTED pSrcBuf : PVOID
GET
pSrcBuf := ADR(nValue);
END_GET
END_PROPERTY

{attribute 'monitoring':='call'}
PROPERTY Value : BOOL
GET
Value := nValue;
END_GET
SET
nValue := Value;

//Trigger a new write cycle
THIS^.bWriteDone 	:= FALSE;
END_SET
END_PROPERTY

END_FUNCTION_BLOCK

// COMPONENTs/CoE-Access/FB_CoE_BYTE
{attribute 'no_explicit_call' := 'Do not call the body - Stick to OOP'}
FUNCTION_BLOCK FB_CoE_BYTE EXTENDS FB_CoE_Base
(* 
   FB_init:
	(	ipCoeConnection := fbCoeConnection, (*each EC-Slave needs one FB_CoE_Connection*)
		nIndex     		:= 16#8010, (* CoE Object Index *)
		nSubIndex  		:= 16#11 (* Subindex of CoE Object *));
 *)
VAR
	{attribute 'hide'}
	nValue : BYTE;
END_VAR

PROPERTY PROTECTED cbBufLen : UDINT
GET
cbBufLen := SIZEOF(nValue);
END_GET
END_PROPERTY

PROPERTY PROTECTED pSrcBuf : PVOID
GET
pSrcBuf := ADR(nValue);
END_GET
END_PROPERTY

{attribute 'monitoring':='call'}
PROPERTY Value : BYTE
GET
Value := nValue;
END_GET
SET
nValue := Value;

//Trigger a new write cycle
THIS^.bWriteDone 	:= FALSE;
END_SET
END_PROPERTY

END_FUNCTION_BLOCK

// COMPONENTs/CoE-Access/FB_CoE_Connection
(* This FB must be instantiated once per EtherCat slave. 
It is used to generate the PLC process image required to read the ADS address + port from the terminal. 
This information is then transferred to the individual FBs for the registers *)
{attribute 'no_explicit_call' := 'Do not call the body - Stick to OOP'}
FUNCTION_BLOCK  FB_CoE_Connection IMPLEMENTS I_AdsAddr
VAR
	AdsAddr AT %I* : AMSADDR;
END_VAR

{attribute 'monitoring':='call'}
PROPERTY Mapped : BOOL
GET
VAR
	bNotMapped : BOOL;
END_VAR
bNotMapped := F_GetMappingStatus(ADR(THIS^.AdsAddr), SIZEOF(THIS^.AdsAddr)) <> EPlcMappingStatus.MS_Mapped;

Mapped := NOT bNotMapped;
END_GET
END_PROPERTY

{attribute 'monitoring':='call'}
PROPERTY NetId : T_AmsNetID
GET
//Convert number to string
NetId := F_CreateAmsNetId( AdsAddr.netId );
END_GET
END_PROPERTY

{attribute 'monitoring':='call'}
PROPERTY Port : WORD
GET
Port := AdsAddr.port;
END_GET
END_PROPERTY

END_FUNCTION_BLOCK

// COMPONENTs/CoE-Access/FB_CoE_UDINT
{attribute 'no_explicit_call' := 'Do not call the body - Stick to OOP'}
FUNCTION_BLOCK FB_CoE_UDINT EXTENDS FB_CoE_Base
(* 
   FB_init:
	(	ipCoeConnection := fbCoeConnection, (*each EC-Slave needs one FB_CoE_Connection*)
		nIndex     		:= 16#8010, (* CoE Object Index *)
		nSubIndex  		:= 16#11 (* Subindex of CoE Object *));
 *)
VAR
	{attribute 'hide'}
	nValue : UDINT;
END_VAR

PROPERTY PROTECTED cbBufLen : UDINT
GET
cbBufLen := SIZEOF(nValue);
END_GET
END_PROPERTY

PROPERTY PROTECTED pSrcBuf : PVOID
GET
pSrcBuf := ADR(nValue);
END_GET
END_PROPERTY

{attribute 'monitoring':='call'}
PROPERTY Value : UDINT
GET
Value := nValue;
END_GET
SET
nValue := Value;

//Trigger a new write cycle
THIS^.bWriteDone 	:= FALSE;
END_SET
END_PROPERTY

END_FUNCTION_BLOCK

// COMPONENTs/CoE-Access/FB_CoE_UINT
{attribute 'no_explicit_call' := 'Do not call the body - Stick to OOP'}
FUNCTION_BLOCK FB_CoE_UINT EXTENDS FB_CoE_Base
(* 
   FB_init:
	(	ipCoeConnection := fbCoeConnection, (*each EC-Slave needs one FB_CoE_Connection*)
		nIndex     		:= 16#8010, (* CoE Object Index *)
		nSubIndex  		:= 16#11 (* Subindex of CoE Object *));
 *)
VAR
	{attribute 'hide'}
	nValue : UINT;
END_VAR

PROPERTY PROTECTED cbBufLen : UDINT
GET
cbBufLen := SIZEOF(nValue);
END_GET
END_PROPERTY

PROPERTY PROTECTED pSrcBuf : PVOID
GET
pSrcBuf := ADR(nValue);
END_GET
END_PROPERTY

{attribute 'monitoring':='call'}
PROPERTY Value : UINT
GET
Value := nValue;
END_GET
SET
nValue := Value;

//Trigger a new write cycle
THIS^.bWriteDone 	:= FALSE;
END_SET
END_PROPERTY

END_FUNCTION_BLOCK

// COMPONENTs/EtherCatDiag/Subobject/FB_EtherCatSlaveDiag
FUNCTION_BLOCK FB_EtherCatSlaveDiag EXTENDS FB_CH_Object
VAR
	//data of this slave
	{attribute 'hide'}    
	stEcSlaveConfigData : ST_EcSlaveConfigData;
	{attribute 'hide'}    
	stEtherCatMasterNetID : AMSNETID;
	{attribute 'hide'}    
	stDeviceAmsAddr : AMSADDR;
	{attribute 'hide'}    
	nSeqRead : UINT;
	{attribute 'hide'}  
	nSeqWrite : UINT;
	{attribute 'hide'}    
	bDoWriteState : BOOL;
	{attribute 'hide'}    
	bReadWasSucessfullAtLeadtOnce : BOOL;
	{attribute 'hide'}    
	fbEcGetSlaveState : Tc2_EtherCAT.FB_EcGetSlaveState;
	{attribute 'hide'}    
	fbEcSetSlaveState : Tc2_EtherCAT.FB_EcReqSlaveState;
	{attribute 'hide'}    
END_VAR

METHOD PROTECTED AlarmHandling : BOOL
VAR	
	bErrorNotInOp 	: BOOL;
	bErrorNoCom 	: BOOL;
	bWarningMissingLink : BOOL;
	sPort		: STRING(2);
END_VAR
VAR_INST
	{attribute 'hide'}  
	fbAlarmNotInOpMode : FB_TcAlarm;
	{attribute 'hide'}  
	fbAlarmNotPresent : FB_TcAlarm;
	{attribute 'hide'}  
	fbWarningMissingLink : FB_TcAlarm;
	{attribute 'hide'}  
	sPortLinkMissingOld : STRING(2); 
END_VAR
IF THIS^.fbEcGetSlaveState.bBusy OR THIS^.fbEcGetSlaveState.bError OR NOT bReadWasSucessfullAtLeadtOnce THEN
	// Do not check if read is active	
	RETURN;
	
ELSE
	bErrorNoCom := THIS^.StateBits.bLinkNotPresent;
	bErrorNotInOp := NOT THIS^.StateBits.bOp AND NOT bErrorNoCom;
	bWarningMissingLink := THIS^.StateBits.bLinkMissing;
	
	IF THIS^.StateBits.bPortA THEN
		sPort := 'A';
	ELSIF THIS^.StateBits.bPortB THEN
		sPort := 'B';
	ELSIF THIS^.StateBits.bPortC THEN
		sPort := 'C';
	ELSIF THIS^.StateBits.bPortD THEN
		sPort := 'D';
	ELSE
		sPort := '';	
		bWarningMissingLink := FALSE;
	END_IF
	
	
	
END_IF

//EcNotInOP
IF bErrorNotInOp AND NOT fbAlarmNotInOpMode.bRaised THEN
	fbAlarmNotInOpMode.CreateEx(stEventEntry := TC_EVENTS.CHALET_Base_Events.EcNotInOP, ipSourceInfo := THIS^.fbSourceInfo, bWithConfirmation := FALSE);
	//EtherCAT device {0} is not in OP Mode
	fbAlarmNotInOpMode.ipArguments.Clear().AddStringByValue(THIS^.Name);
	fbAlarmNotInOpMode.Raise(0);

ELSIF NOT bErrorNotInOp AND fbAlarmNotInOpMode.bRaised THEN
	fbAlarmNotInOpMode.Clear(0,0);
END_IF

//EcLinkStateNotPresent
IF bErrorNoCom AND NOT fbAlarmNotPresent.bRaised THEN
	fbAlarmNotPresent.CreateEx(stEventEntry := TC_EVENTS.CHALET_Base_Events.EcLinkStateNotPresent, ipSourceInfo := THIS^.fbSourceInfo, bWithConfirmation := FALSE);
	//No EtherCAT communication with the EtherCAT device {0}
	fbAlarmNotPresent.ipArguments.Clear().AddStringByValue(THIS^.Name);
	fbAlarmNotPresent.Raise(0);

ELSIF NOT bErrorNoCom AND fbAlarmNotPresent.bRaised THEN
	fbAlarmNotPresent.Clear(0,0);
END_IF

//EcMissingLink
IF bWarningMissingLink AND NOT fbWarningMissingLink.bRaised THEN
	fbWarningMissingLink.CreateEx(stEventEntry := TC_EVENTS.CHALET_Base_Events.EcMissingLink, ipSourceInfo := THIS^.fbSourceInfo, bWithConfirmation := FALSE);
	//EtherCAT Device {0} is missing connection on Port {1}
	fbWarningMissingLink.ipArguments.Clear().AddStringByValue(THIS^.Name).AddStringByValue(sPort);
	fbWarningMissingLink.Raise(0);
	sPortLinkMissingOld := sPort;

ELSIF (NOT bWarningMissingLink OR sPortLinkMissingOld <> sPort) AND fbWarningMissingLink.bRaised THEN
	fbWarningMissingLink.Clear(0,0);
END_IF
END_METHOD

{attribute 'monitoring':='call'}
PROPERTY DeviceAmsAddr : AMSADDR
GET

DeviceAmsAddr :=  stDeviceAmsAddr;
END_GET
END_PROPERTY

{attribute 'monitoring':='call'}
PROPERTY DeviceType : STRING(15)
GET
DeviceType := THIS^.stEcSlaveConfigData.sType;
END_GET
END_PROPERTY

{attribute 'monitoring':='call'}
PROPERTY Name : STRING(31)
GET
Name := THIS^.stEcSlaveConfigData.sName;
END_GET
END_PROPERTY

METHOD SetConfig : BOOL
VAR_INPUT
	stEtherCatMasterNetID : AMSNETID;
	stEcSlaveConfigData : ST_EcSlaveConfigData;
END_VAR
THIS^.stEcSlaveConfigData := stEcSlaveConfigData;
THIS^.stEtherCatMasterNetID := stEtherCatMasterNetID;

//Set name in TC3_Eventlogger
THIS^.fbSourceInfo.sName := stEcSlaveConfigData.sName;

//Same as master
stDeviceAmsAddr.netId := THIS^.stEtherCatMasterNetID;

//Set Port
stDeviceAmsAddr.port := THIS^.stEcSlaveConfigData.nAddr;
END_METHOD

{attribute 'monitoring':='call'}
PROPERTY State : E_EtherCatState
GET
VAR
	stStateBits : ST_EcSlaveStateBitsEx;
END_VAR
stStateBits := THIS^.StateBits;

//Convert bit to enum
IF stStateBits.bOp THEN
	State := E_EtherCatState.Op;
	
ELSIF stStateBits.bSafeOp THEN
	State := E_EtherCatState.SafeOp;
	
ELSIF stStateBits.bPreop THEN
	State := E_EtherCatState.PreOp;
	
ELSIF stStateBits.bInit THEN
	State := E_EtherCatState.Init;
	
ELSIF stStateBits.bError THEN
	State := E_EtherCatState.Error;
	
ELSIF stStateBits.bBootStrap THEN
	State := E_EtherCatState.BootStrap;
	
ELSIF stStateBits.bDisabled THEN
	State := E_EtherCatState.Disabled;
	
	
ELSE
	//Unknown
	State := E_EtherCatState.Unknown;	
END_IF
END_GET
SET
IF State = E_EtherCatState.Unknown THEN
	//Not allowed
	RETURN;
END_IF



CASE State OF
	E_EtherCatState.Op:
		fbEcSetSlaveState.state := EC_DEVICE_STATE_OP;
		bDoWriteState := TRUE;
	
	E_EtherCatState.SafeOp:
		fbEcSetSlaveState.state := EC_DEVICE_STATE_SAFEOP;
		bDoWriteState := TRUE;
    
	E_EtherCatState.PreOp:
		fbEcSetSlaveState.state := EC_DEVICE_STATE_PREOP;
		bDoWriteState := TRUE;
    
	E_EtherCatState.Init:
		fbEcSetSlaveState.state := EC_DEVICE_STATE_INIT;
		bDoWriteState := TRUE;
    
	E_EtherCatState.Error:
		fbEcSetSlaveState.state := EC_DEVICE_STATE_ERROR;
		bDoWriteState := TRUE;
    
	E_EtherCatState.BootStrap:
		fbEcSetSlaveState.state := EC_DEVICE_STATE_BOOTSTRAP;
		bDoWriteState := TRUE; 

END_CASE
END_SET
END_PROPERTY

{attribute 'monitoring':='call'}
PROPERTY StateBits : REFERENCE TO ST_EcSlaveStateBitsEx
GET
VAR
	stSlaveStateSource : ST_EcSlaveState;
	stSlaveStateDest : ST_EcSlaveStateBitsEx;
	
	bLinkStateOk : BOOL;
END_VAR
stSlaveStateSource := THIS^.fbEcGetSlaveState.state;


//deviceState
stSlaveStateDest.bInit 			:= (stSlaveStateSource.deviceState = EC_DEVICE_STATE_INIT);
stSlaveStateDest.bBootStrap 	:= (stSlaveStateSource.deviceState = EC_DEVICE_STATE_BOOTSTRAP);
stSlaveStateDest.bPreop 		:= (stSlaveStateSource.deviceState = EC_DEVICE_STATE_PREOP);
stSlaveStateDest.bSafeOp 		:= (stSlaveStateSource.deviceState = EC_DEVICE_STATE_SAFEOP);
stSlaveStateDest.bOp 			:= (stSlaveStateSource.deviceState = EC_DEVICE_STATE_OP);
stSlaveStateDest.bError 		:= (stSlaveStateSource.deviceState = EC_DEVICE_STATE_ERROR);
stSlaveStateDest.bInvVPRS 		:= (stSlaveStateSource.deviceState = EC_DEVICE_STATE_INVALID_VPRS);
stSlaveStateDest.bInitCmdError 	:= (stSlaveStateSource.deviceState = EC_DEVICE_STATE_INITCMD_ERROR);
stSlaveStateDest.bDisabled 		:= (stSlaveStateSource.deviceState = EC_DEVICE_STATE_DISABLED);


//linkState multiple bits
bLinkStateOk 						:= (stSlaveStateSource.linkState AND EC_LINK_STATE_OK) > 0;
stSlaveStateDest.bLinkNotPresent 	:= (stSlaveStateSource.linkState AND EC_LINK_STATE_NOT_PRESENT) > 0;
stSlaveStateDest.bLinkWithoutComm 	:= (stSlaveStateSource.linkState AND EC_LINK_STATE_LINK_WITHOUT_COMM) > 0;
stSlaveStateDest.bLinkMissing 		:= (stSlaveStateSource.linkState AND EC_LINK_STATE_MISSING_LINK) > 0;
stSlaveStateDest.bAdditionalLink 	:= (stSlaveStateSource.linkState AND EC_LINK_STATE_ADDITIONAL_LINK) > 0;
stSlaveStateDest.bPortA 			:= (stSlaveStateSource.linkState AND EC_LINK_STATE_PORT_A) > 0;
stSlaveStateDest.bPortB 			:= (stSlaveStateSource.linkState AND EC_LINK_STATE_PORT_B) > 0;
stSlaveStateDest.bPortC 			:= (stSlaveStateSource.linkState AND EC_LINK_STATE_PORT_C) > 0;
stSlaveStateDest.bPortD 			:= (stSlaveStateSource.linkState AND EC_LINK_STATE_PORT_D) > 0;


StateBits REF= stSlaveStateDest;
END_GET
END_PROPERTY

METHOD Update : HRESULT
VAR
END_VAR
CASE nSeqRead OF
	0: //start read state 
		fbEcGetSlaveState.bExecute := TRUE;
		nSeqRead := 1;
		
	1: //wait
		IF NOT fbEcGetSlaveState.bBusy THEN
			fbEcGetSlaveState.bExecute := FALSE;
			nSeqRead := 0;
		END_IF
		IF NOT fbEcGetSlaveState.bBusy AND NOT fbEcGetSlaveState.bError THEN
			bReadWasSucessfullAtLeadtOnce := TRUE;
		END_IF
		
		
		
		
		
END_CASE

CASE nSeqWrite OF
	0: //start write state request
		IF bDoWriteState THEN
			fbEcSetSlaveState.bExecute := TRUE;
			nSeqWrite := 1;
		END_IF
		
	1: //wait
		IF NOT fbEcSetSlaveState.bBusy THEN
			fbEcSetSlaveState.bExecute := FALSE;
			nSeqWrite := 0;
		END_IF
		IF NOT fbEcSetSlaveState.bBusy AND NOT fbEcSetSlaveState.bError THEN
			bDoWriteState := FALSE;
		END_IF
END_CASE


//Call subroutine
AlarmHandling();




fbEcGetSlaveState(
	sNetId:= Tc2_System.F_CreateAmsNetId(nIds:= stDeviceAmsAddr.netId), 
	nSlaveAddr:= stDeviceAmsAddr.port);
	
fbEcSetSlaveState(
	sNetId:= Tc2_System.F_CreateAmsNetId(nIds:= stDeviceAmsAddr.netId), 
	nSlaveAddr:= stDeviceAmsAddr.port);
END_METHOD

END_FUNCTION_BLOCK

// COMPONENTs/EtherCatDiag/Subobject/I_EtherCatSlaveDiag
INTERFACE I_EtherCatSlaveDiag EXTENDS I_CH_Object

{attribute 'monitoring':='call'}
PROPERTY DeviceAmsAddr : AMSADDR
GET
END_GET
END_PROPERTY

{attribute 'monitoring':='call'}
PROPERTY DeviceType : STRING(15)
GET
END_GET
END_PROPERTY

{attribute 'monitoring':='call'}
PROPERTY Name : STRING(31)
GET
END_GET
END_PROPERTY

{attribute 'monitoring':='call'}
PROPERTY State : E_EtherCatState
GET
END_GET
SET
END_SET
END_PROPERTY

{attribute 'monitoring':='call'}
PROPERTY StateBits : REFERENCE TO ST_EcSlaveStateBitsEx
GET
END_GET
END_PROPERTY

END_INTERFACE

// COMPONENTs/EtherCatDiag/FB_EtherCatMasterDiag
{attribute 'no_explicit_call' := 'Do not call the body - Stick to OOP'}
(* This FB generates an array with all XTS motor modules. These are now checked cyclically one after the other to see whether the EtherCAT slave controller is in OP mode *)
FUNCTION_BLOCK FB_EtherCatMasterDiag EXTENDS FB_CH_Object
VAR
	//Link to AMS NET ID of EtherCAT master
	EtherCatMasterNetID AT %I* : AMSNETID;
	fbEtherCatSlaveDiag : ARRAY [0..(BaseParameterlist.MAX_OBJECTS)] OF FB_EtherCatSlaveDiag;

	
	{attribute 'hide'}  
	fbListOfEtherCatSlaves : FB_CH_List;
	
	{attribute 'hide'}  
	bInitDone : BOOL;

	{attribute 'hide'}  
	fbGetConfSlaves : FB_EcGetConfSlaves;


	{attribute 'hide'}  
	stEcSlaveConfigData : ARRAY [0..(BaseParameterlist.MAX_OBJECTS)] OF ST_EcSlaveConfigData;
END_VAR

METHOD Initialize : HRESULT
VAR
	nIdx : UDINT;
	stVarInfo : __SYSTEM.VAR_INFO;
END_VAR
VAR_INST
	{attribute 'hide'}	
	nInitSeq : UINT;
	//This error cannot be reset. Requires a reset cold
	{attribute 'hide'}	
	fbInitError : FB_TcAlarm;
END_VAR
// Check if link to MC-Mover is mapped
IF NOT THIS^.Mapped THEN
	IF NOT fbInitError.bRaised THEN 
		//This error cannot be reset. Requires a reset cold
		fbInitError.CreateEx(stEventEntry:=TC_EVENTS.CHALET_Base_Events.VariableLinkMissing, ipSourceInfo := THIS^.fbSourceInfo, bWithConfirmation := FALSE);
		stVarInfo := __VARINFO(EtherCatMasterNetID);
		fbInitError.ipArguments.AddString(stVarInfo.Symbol);
		fbInitError.Raise(0);
	END_IF
	Initialize := E_FAIL;
	RETURN;
END_IF


CASE nInitSeq OF
	
	0: //Validate condition to start scan
		IF THIS^.Mapped AND EtherCatMasterNetID[5] <> 0 THEN
			fbGetConfSlaves.sNetId := Tc2_System.F_CreateAmsNetId(nIds:= EtherCatMasterNetID);
			nInitSeq := 1;
		END_IF
	
	1: //Start scan
		fbGetConfSlaves.bExecute := TRUE;	
		nInitSeq := 2;

	2: //Wait for done or error
		IF NOT fbGetConfSlaves.bBusy THEN
			nInitSeq := 3;
			FOR nIdx := 0 TO BaseParameterlist.MAX_OBJECTS DO
				IF stEcSlaveConfigData[nIdx].nAddr <> 0 THEN
					//handover info to fb for each slave
					fbEtherCatSlaveDiag[nIdx].SetConfig(stEcSlaveConfigData := stEcSlaveConfigData[nIdx], 
														stEtherCatMasterNetID := THIS^.EtherCatMasterNetID);
					//add to list
					fbListOfEtherCatSlaves.AddObject(fbEtherCatSlaveDiag[nIdx]);
				END_IF
			END_FOR
			
			nInitSeq := 3;
		END_IF

	3: //Init List of slave diag FBs until S_OK;
		IF fbListOfEtherCatSlaves.Initialize() = S_OK THEN
			bInitDone := TRUE;
			nInitSeq := 999;
		END_IF
		
END_CASE


//Cyclic update
fbGetConfSlaves(pArrEcConfSlaveInfo := ADR(stEcSlaveConfigData), cbBufLen := SIZEOF(stEcSlaveConfigData));
END_METHOD

{attribute 'monitoring':='call'}
PROPERTY Initialized : BOOL
GET
Initialized := bInitDone;
END_GET
END_PROPERTY

{attribute 'monitoring':='call'}
PROPERTY ListOfDevices : I_CH_List
GET
ListOfDevices := THIS^.fbListOfEtherCatSlaves;
END_GET
END_PROPERTY

{attribute 'monitoring':='call'}
PROPERTY Mapped : BOOL //Mapping to EtherCatMaster AMSNETID
GET
VAR
	bIoPlcNotMapped 	: BOOL;
END_VAR
bIoPlcNotMapped := F_GetMappingStatus(ADR(THIS^.EtherCatMasterNetID), SIZEOF(THIS^.EtherCatMasterNetID)) <> EPlcMappingStatus.MS_Mapped;

Mapped := NOT bIoPlcNotMapped;
END_GET
END_PROPERTY

{attribute 'monitoring':='call'}
PROPERTY NumerOfDevice : UDINT
GET
NumerOfDevice := fbListOfEtherCatSlaves.Size;
END_GET
END_PROPERTY

METHOD Update : HRESULT
VAR
END_VAR
//Force to do init
IF NOT THIS^.Initialized THEN
	Initialize();
	RETURN;
END_IF



//Update whole list but only one slave at once
IF fbListOfEtherCatSlaves.HasNextObject() THEN
	fbListOfEtherCatSlaves.GetNextObject().Update();
ELSE
	fbListOfEtherCatSlaves.ResetIterator();
END_IF
END_METHOD

END_FUNCTION_BLOCK

// COMPONENTs/Feedback/FB_CH_Feedback
FUNCTION_BLOCK FB_CH_Feedback IMPLEMENTS I_CH_Feedback
VAR
    {attribute 'hide'}
    _hr : HRESULT;
    {attribute 'hide'}
    _activeCommand : STRING;
    {attribute 'hide'}
    _lastCommandAccepted : BOOL;
    {attribute 'hide'}
    fbAlarm : Tc3_EventLogger.FB_TcAlarm;	
	{attribute 'hide'}
	nOldErrorId : UDINT; //last cycle
	{attribute 'hide'}
	bOldBusy	: BOOL; //last cycle
	{attribute 'hide'}
	//Optional. If interface is <>0 a Error is automatic written in TC3_Eventlogger
	ipSourceInfo : I_TcSourceInfo;
END_VAR

{attribute 'monitoring' := 'call'}
PROPERTY ActiveCommand : STRING;
GET
ActiveCommand := THIS^._ActiveCommand;
END_GET
SET
THIS^._ActiveCommand 		:= ActiveCommand;
END_SET
END_PROPERTY

{attribute 'monitoring' := 'call'}
(* Indicates a busy command, i.e. command is being processed, waiting for execution, or already executing (= also active). *)
PROPERTY Busy : BOOL
GET
Busy := (THIS^._hr = S_PENDING);
END_GET
SET
IF Busy THEN
	THIS^._hr := S_PENDING;
END_IF

THIS^.UpdateEventlogger();
END_SET
END_PROPERTY

{attribute 'monitoring' := 'call'}
(* Indicates the command is done, i.e. execution of the command finished successfully. *)
PROPERTY Done : BOOL
GET
Done := NOT THIS^.Busy AND NOT THIS^.Error;
END_GET
SET
IF Done THEN
	THIS^._hr := S_OK;
END_IF


THIS^.UpdateEventlogger();
END_SET
END_PROPERTY

{attribute 'monitoring' := 'call'}
(* Indicates the command has an error. *)
PROPERTY Error : BOOL
GET
Error := FAILED(THIS^._hr);
END_GET
END_PROPERTY

{attribute 'monitoring' := 'call'}
(* Indicates the error id of the command error. *)
PROPERTY ErrorId : UDINT
GET
ErrorId := DWORD_TO_UDINT(DINT_TO_DWORD(THIS^._hr) AND 16#0000FFFF); //only return the last two byte with the error Id

//515 means busy and is not an Error
IF ErrorId = 515 THEN
	ErrorId := 0;
END_IF
END_GET
SET
VAR
	//A failed execution is indicated by a NEGATIVE code, or in hexadecimal notation the first digit is >= 8.
	nErrorCodeSign : UDINT := 2#10000000000000000000000000000000;
END_VAR
IF ErrorId <> 0 THEN
	//Bitwise OR
	THIS^._hr := DWORD_TO_DINT(TO_DWORD(nErrorCodeSign) OR TO_DWORD(ErrorId));
END_IF


THIS^.UpdateEventlogger();
END_SET
END_PROPERTY

METHOD FB_init : BOOL
VAR_INPUT
	bInitRetains : BOOL; // if TRUE, the retain variables are initialized (warm start / cold start)
	bInCopyCode : BOOL;  // if TRUE, the instance afterwards gets moved into the copy code (online change)
	
	//Optional. If interface is <>0 a Error is automatic written in TC3_Eventlogger
	ipSourceInfo : I_TcSourceInfo;
END_VAR
THIS^.ipSourceInfo := ipSourceInfo;
END_METHOD

{attribute 'monitoring' := 'call'}
PROPERTY HR : HRESULT
GET
HR := THIS^._hr;
END_GET
SET
THIS^._hr := HR;

THIS^.UpdateEventlogger();
END_SET
END_PROPERTY

{attribute 'monitoring' := 'call'}
PROPERTY LastCommandAccepted : BOOL
GET
LastCommandAccepted := THIS^._lastCommandAccepted;
END_GET
SET
THIS^._lastCommandAccepted := LastCommandAccepted;
END_SET
END_PROPERTY

METHOD PROTECTED UpdateEventlogger : BOOL
VAR
	nHR : DWORD;
END_VAR
IF THIS^.ipSourceInfo = 0 THEN
	//No TC3_Eventlogger alarm if interface is empty
	RETURN;
END_IF


//New error, raise alarm
IF (THIS^.ErrorId <> THIS^.nOldErrorId) AND THIS^.Error THEN
	THIS^.fbAlarm.Clear(0,0);
	THIS^.fbAlarm.CreateEx(stEventEntry := TC_EVENTS.CHALET_Base_Events.FeedbackErrorCmd, ipSourceInfo := THIS^.ipSourceInfo, bWithConfirmation:= FALSE);
	//Error in feedback command {0} error id {1}
	
	//Convert to DWORD
	nHR := TO_DWORD(THIS^.HR);
	
	//Try to get some more details about error id
	IF THIS^.HR = E_FAIL THEN
		THIS^.fbAlarm.ipArguments.Clear().AddStringByValue(THIS^.ActiveCommand).AddStringByValue('E_FAIL');
		
	ELSIF ((nHR AND 16#FFFF_FF00) = 16#9811_0000) THEN
		THIS^.fbAlarm.ipArguments.Clear().AddStringByValue(THIS^.ActiveCommand).AddUDInt(THIS^.ErrorId).AddEventReferenceIdGuid(nEventId := THIS^.ErrorId, EventClass := TC_EVENT_CLASSES.TcSystemEventClass);
		;//Global error codes
			
	ELSIF ((nHR AND 16#FFFF_FF00) = 16#9811_0500) THEN
		THIS^.fbAlarm.ipArguments.Clear().AddStringByValue(THIS^.ActiveCommand).AddUDInt(THIS^.ErrorId).AddEventReferenceIdGuid(nEventId := THIS^.ErrorId, EventClass := TC_EVENT_CLASSES.TcRouterEventClass);
		;//Router error codes
			
	ELSIF ((nHR AND 16#FFFF_FF00) = 16#9811_0700) THEN
		THIS^.fbAlarm.ipArguments.Clear().AddStringByValue(THIS^.ActiveCommand).AddUDInt(THIS^.ErrorId).AddEventReferenceIdGuid(nEventId := THIS^.ErrorId, EventClass := TC_EVENT_CLASSES.TcGeneralAdsEventClass);
		;//General ADS errors
			
	ELSIF ((nHR AND 16#FFFF_FF00) = 16#9811_1000) THEN
		THIS^.fbAlarm.ipArguments.Clear().AddStringByValue(THIS^.ActiveCommand).AddUDInt(THIS^.ErrorId).AddEventReferenceIdGuid(nEventId := THIS^.ErrorId, EventClass := TC_EVENT_CLASSES.TcRTimeEventClass);
		;//RTime error codes
	
	ELSE
		THIS^.fbAlarm.ipArguments.Clear().AddStringByValue(THIS^.ActiveCommand).AddUDInt(THIS^.ErrorId);
	END_IF
	
	THIS^.fbAlarm.Raise(0);

	
//Busy, raise info
ELSIF (THIS^.Busy <> THIS^.bOldBusy) AND THIS^.Busy AND BaseParameterlist.B_WRITE_INFO_FEEDBACK_BUSY THEN
	THIS^.fbAlarm.Clear(0,0);
	THIS^.fbAlarm.CreateEx(stEventEntry := TC_EVENTS.CHALET_Base_Events.FeedbackBusy, ipSourceInfo := THIS^.ipSourceInfo, bWithConfirmation:= FALSE);
	THIS^.fbAlarm.ipArguments.Clear().AddStringByValue(THIS^.ActiveCommand);
	THIS^.fbAlarm.Raise(0);
	
//No error, clear alarm	
ELSIF NOT THIS^.Error AND NOT (THIS^.Busy AND BaseParameterlist.B_WRITE_INFO_FEEDBACK_BUSY) THEN
	THIS^.fbAlarm.Clear(0,0);
END_IF

THIS^.nOldErrorId 	:= THIS^.ErrorId;
THIS^.bOldBusy 		:= THIS^.Busy;
END_METHOD

END_FUNCTION_BLOCK

// COMPONENTs/Feedback/I_CH_Feedback
INTERFACE I_CH_Feedback

{attribute 'monitoring' := 'call'}
PROPERTY ActiveCommand : STRING;
GET
END_GET
END_PROPERTY

{attribute 'monitoring' := 'call'}
(* Indicates a busy command, i.e. command is being processed, waiting for execution, or already executing (= also active). *)
PROPERTY Busy : BOOL
GET
END_GET
END_PROPERTY

{attribute 'monitoring' := 'call'}
(* Indicates the command is done, i.e. execution of the command finished successfully. *)
PROPERTY Done : BOOL
GET
END_GET
END_PROPERTY

{attribute 'monitoring' := 'call'}
(* Indicates the command has an error. *)
PROPERTY Error : BOOL
GET
END_GET
END_PROPERTY

{attribute 'monitoring' := 'call'}
(* Indicates the error id of the command error. *)
PROPERTY ErrorId : UDINT
GET
END_GET
END_PROPERTY

{attribute 'monitoring' := 'call'}
PROPERTY HR : HRESULT
GET
END_GET
END_PROPERTY

{attribute 'monitoring' := 'call'}
PROPERTY LastCommandAccepted : BOOL
GET
END_GET
END_PROPERTY

END_INTERFACE

// COMPONENTs/HR/CheckNotOk
FUNCTION CheckNotOk : BOOL
VAR_INPUT
	hr : HRESULT;
END_VAR

CheckNotOk := (hr <> S_OK);

END_FUNCTION

// COMPONENTs/HR/CheckOk
FUNCTION CheckOk : BOOL
VAR_INPUT
	hr : HRESULT;
END_VAR

CheckOk := (hr = S_OK);

END_FUNCTION

// COMPONENTs/F_Convert32InPastTo64Bit
FUNCTION F_Convert32InPastTo64Bit : T_DCTIME64
VAR_INPUT
	nTimeInPast32 : T_DCTIME32;
END_VAR
VAR
	nCurDcTaskTime :T_DCTIME;
	nNextOutputStartTime_DCTIME :T_DCTIME;
END_VAR

//Convert 32bit (max 4.2sec) time format in 64bit (584year)
nCurDcTaskTime := F_GetCurDcTaskTime();
nNextOutputStartTime_DCTIME.dwHighPart := nCurDcTaskTime.dwHighPart;
nNextOutputStartTime_DCTIME.dwLowPart := nTimeInPast32;

//StartTimeNextOutput is allways in the past
IF nTimeInPast32 > nCurDcTaskTime.dwLowPart THEN 
	nNextOutputStartTime_DCTIME.dwHighPart := nNextOutputStartTime_DCTIME.dwHighPart - 1;
END_IF

//Convert in  64bit datetype
F_Convert32InPastTo64Bit:= DCTIME_TO_DCTIME64(nNextOutputStartTime_DCTIME);

END_FUNCTION
